// TIA Portal project "Pump Cycling" (V17)
// Pump Cycling
// Turn ON a pump for 10 sec, then OFF for 20 seconds and repeats this cycle

(* hardware
DEVICE "S7-1200 station_1"  S7-1200 Station
   slot 0: "Rack_0"  S7-1200 Rack  Rack  V1.0
   slot 1: "PLC_1"  CPU 1211C AC/DC/Rly  6ES7 211-1BE40-0XB0  V4.5
*)

// ===== PLC "PLC_1"  CPU 1211C AC/DC/Rly =====

VAR_GLOBAL   // PLC tag table "Default tag table"
   "PB" AT %I0.0 : Bool;
   "Pump ON" AT %Q0.0 : Bool;
   "Tag_1" AT %M0.0 : Bool;
END_VAR

// folder: System blocks/Program resources

DATA_BLOCK "IEC_Timer_0_DB"   // DB1
{ S7_Optimized_Access := 'TRUE' }
AUTHOR : Simatic
FAMILY : IEC
NAME : IEC_TMR
VERSION : 1.0
// stored: InstanceOfName IEC_TIMER
"IEC_TIMER"
BEGIN
END_DATA_BLOCK

DATA_BLOCK "IEC_Timer_0_DB_1"   // DB2
{ S7_Optimized_Access := 'TRUE' }
AUTHOR : Simatic
FAMILY : IEC
NAME : IEC_TMR
VERSION : 1.0
// stored: InstanceOfName IEC_TIMER
"IEC_TIMER"
BEGIN
END_DATA_BLOCK

// folder: (top level)

ORGANIZATION_BLOCK "Main"   // OB1, LAD, ProgramCycle
TITLE = "Main Program Sweep (Cycle)"
{ S7_Optimized_Access := 'TRUE' }
VERSION : 0.1
   VAR_INPUT
      Initial_Call : Bool;   // Initial call of this OB
      Remanence : Bool;   // =True, if remanent data are available
   END_VAR
   VAR_TEMP   // added for the SCL form of the ladder/FBD networks
      _w1 : Bool;
   END_VAR
BEGIN

REGION Network 1
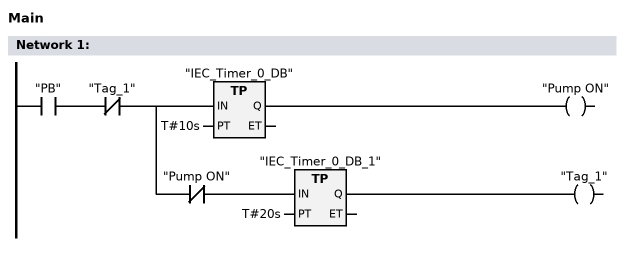
   #_w1 := "PB" AND NOT "Tag_1";
   "IEC_Timer_0_DB".TP(IN := #_w1, PT := T#10s);
   "Pump ON" := "IEC_Timer_0_DB".Q;
   "IEC_Timer_0_DB_1".TP(IN := #_w1 AND NOT "Pump ON", PT := T#20s);
   "Tag_1" := "IEC_Timer_0_DB_1".Q;
END_REGION
END_ORGANIZATION_BLOCK